PROGRAM MAIN
VAR
END_VAR

END_PROGRAM

(* stored: Version 1.1.0.1
   POU MAIN: Id {bf34bab7-6eef-432e-ab84-9c3203dbf679} *)
